PROGRAM MAIN
VAR
	i :WORD;
END_VAR

i := i +1;

END_PROGRAM

(* stored: Version 1.1.0.1
   POU MAIN: Id {cbbb1d50-43c6-4340-9a0c-b36c70a0cffd}, SpecialFunc None *)
